FUNCTION_BLOCK Movement_Controller (* Composite Function Block Type *)
  (* Standard: 61499-2 *)
  (* Version 0.0, 9/23/2026, macie, Schneider Electric, template *)
  PACKAGE Main;
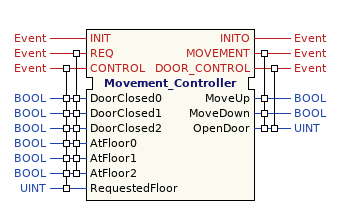
  EVENT_INPUT
    INIT;
    REQ WITH DoorClosed0, DoorClosed1, DoorClosed2, AtFloor0, AtFloor1, AtFloor2; (* Normal Execution Request *)
    CONTROL WITH DoorClosed0, DoorClosed1, DoorClosed2, AtFloor0, AtFloor1, AtFloor2, RequestedFloor;
  END_EVENT
  EVENT_OUTPUT
    INITO;
    MOVEMENT WITH MoveUp, MoveDown, OpenDoor; (* Execution Confirmation *)
    DOOR_CONTROL WITH OpenDoor;
  END_EVENT
  VAR_INPUT
    DoorClosed0 : BOOL; (* Input event qualifier *)
    DoorClosed1 : BOOL;
    DoorClosed2 : BOOL;
    AtFloor0 : BOOL;
    AtFloor1 : BOOL;
    AtFloor2 : BOOL;
    RequestedFloor : UINT;
  END_VAR
  VAR_OUTPUT
    MoveUp : BOOL := FALSE; (* Output event qualifier *)
    MoveDown : BOOL := FALSE;
    OpenDoor : UINT;
  END_VAR
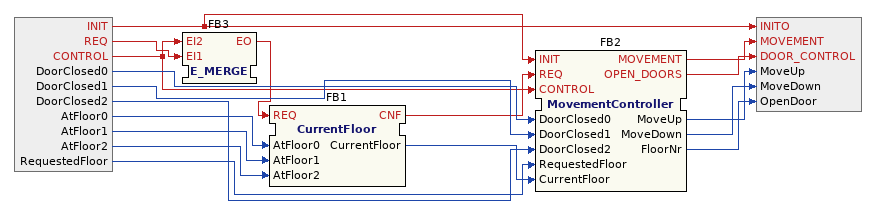
  FBS
    FB2 : MovementController;
    FB1 : CurrentFloor;
    FB3 : E_MERGE;
  END_FBS
  EVENT_CONNECTIONS
    FB2.MOVEMENT TO MOVEMENT;
    FB2.OPEN_DOORS TO DOOR_CONTROL;
    INIT TO FB2.INIT;
    INIT TO INITO;
    FB1.CNF TO FB2.REQ;
    FB3.EO TO FB1.REQ;
    CONTROL TO FB3.EI2;
    REQ TO FB3.EI1;
    CONTROL TO FB2.CONTROL;
  END_CONNECTIONS
  DATA_CONNECTIONS
    DoorClosed0 TO FB2.DoorClosed0;
    DoorClosed1 TO FB2.DoorClosed1;
    DoorClosed2 TO FB2.DoorClosed2;
    RequestedFloor TO FB2.RequestedFloor;
    FB2.FloorNr TO OpenDoor;
    FB2.MoveUp TO MoveUp;
    FB2.MoveDown TO MoveDown;
    AtFloor0 TO FB1.AtFloor0;
    AtFloor1 TO FB1.AtFloor1;
    AtFloor2 TO FB1.AtFloor2;
    FB1.CurrentFloor TO FB2.CurrentFloor;
  END_CONNECTIONS
END_FUNCTION_BLOCK
